(* CODESYS project Beer_machine.project

Project tree, tasks and I/O mapping:
  Device : CODESYS Control Win V3 x64, 3S - Smart Software Solutions GmbH, version 3.5.11.0
    application Application
      libraries: Standard, * (System); VisuDialogs, * (System); Util, * (System)
      task MainTask (cyclic, interval t#10ms, priority 1) calls Plant, Controller
      program Plant [ST]
      global variables GVL
      program Controller [ST]
      visualisation Visualization
      image pool ImagePool
  text list GlobalTextList
  5ce3da45-db07-42e7-a21c-a00fff4ed8f6|C:\Users\mihas\Documents\NSU2026\AM\images\input\MAX.png
  5ce3da45-db07-42e7-a21c-a00fff4ed8f6|C:\Users\mihas\Documents\NSU2026\AM\images\input\beer.png
  5ce3da45-db07-42e7-a21c-a00fff4ed8f6|C:\Users\mihas\Documents\NSU2026\AM\images\input\cigaretes after vki .png
  5ce3da45-db07-42e7-a21c-a00fff4ed8f6|C:\Users\mihas\Documents\NSU2026\AM\images\input\greencard.png
  5ce3da45-db07-42e7-a21c-a00fff4ed8f6|C:\Users\mihas\Documents\NSU2026\AM\images\input\jaguar.png
  5ce3da45-db07-42e7-a21c-a00fff4ed8f6|C:\Users\mihas\Documents\NSU2026\AM\images\input\monster.png
  5ce3da45-db07-42e7-a21c-a00fff4ed8f6|C:\Users\mihas\Documents\NSU2026\AM\images\input\pistol.png
  5ce3da45-db07-42e7-a21c-a00fff4ed8f6|C:\Users\mihas\Documents\NSU2026\AM\images\input\voenbilet.png
  5ce3da45-db07-42e7-a21c-a00fff4ed8f6|C:\Users\fish\AC_Beer_machine\img\input\blue monster.png
  5ce3da45-db07-42e7-a21c-a00fff4ed8f6|C:\Users\fish\AC_Beer_machine\img\input\monster.png
  5ce3da45-db07-42e7-a21c-a00fff4ed8f6|C:\Users\fish\AC_Beer_machine\img\input\red monster.jpg
  5ce3da45-db07-42e7-a21c-a00fff4ed8f6|C:\Users\fish\AC_Beer_machine\img\input\white monster.png
  5ce3da45-db07-42e7-a21c-a00fff4ed8f6|C:\Users\fish\AC_Beer_machine\img\input\yellow monster.png
*)

// Device/Application/GVL
VAR_GLOBAL
END_VAR

// Device/Application/Plant
PROGRAM Plant

VAR CONSTANT
	text_welcome_message : WSTRING(250) := "Здравстсвуйте!!!$nВыберите товар.";
	text_out_of_stock : WSTRING(250) := "Выбранного товара нет в наличии.$nПозвоните в поддержку, чтобы восполнить товар.";
	text_in_stock : WSTRING(250) := "Выбранный товар есть в наличии.$nПодготовка к оплате.";
	text_insert_payment : WSTRING(250) := "Оплатите товар.";
	text_not_enough_money : WSTRING(250) := "Внесите ещё.$nСредств недостаточно.";
	text_stuff_not_dropped : WSTRING(250) := "Товар не сбросился.$n Позвоните в поддержку, чтобы вернули деньги";
	text_mission_completed : WSTRING(250) := "Спасибо за покупку.$nНаслаждайтесь нашей продукцией!";
	
	text_arr : ARRAY[0..6] OF WSTRING(250) := [text_welcome_message, text_out_of_stock, text_in_stock, text_insert_payment, text_not_enough_money, text_stuff_not_dropped, text_mission_completed];
END_VAR

VAR
	cur : BOOL;
	dx : DINT;
	start_time_ms : DINT := TIME_TO_DINT(TIME());
	start_time_text : DINT := TIME_TO_DINT(TIME());
	start_time_angle : DINT := TIME_TO_DINT(TIME());
	angle : DINT := 0;
	j : DINT := 0;
	text_display : WSTRING(250);
	
	
	Drop_control : BOOL := 0;
	
	Drop_control1 : BOOL := 0;
	Drop_control2 : BOOL := 0;
	Drop_control3 : BOOL := 0;
	Drop_control4 : BOOL := 0;
	Drop_control5 : BOOL := 0;

	
	Spring1_prev : BOOL := 0;
	Spring2_prev : BOOL := 0;
	Spring3_prev : BOOL := 0;
	Spring4_prev : BOOL := 0;
	Spring5_prev : BOOL := 0;


	
	

END_VAR

VAR
	
	user: INT;
END_VAR

VAR
	MAX_call : BOOL;
	i : INT;
	
	tratit_bank : BOOL := FALSE;
	kopit_bank : BOOL := FALSE;
	user_bank : UDINT := 0;
	tovar : ARRAY[1..5] OF INT := [3, 3, 3, 3, 3];
END_VAR

// Поворот пружины
IF ((TIME_TO_DINT(TIME())) - start_time_angle) MOD 2000 > (1000 / 25) THEN 
	start_time_angle := TIME_TO_DINT(TIME());
	angle := (angle + 360 / 25) MOD 360;
END_IF

//взаимодействие с банком 
IF kopit_bank THEN
	user_bank := user_bank + 1;
	kopit_bank := FALSE;
END_IF
IF tratit_bank THEN
	IF user_bank > 0 THEN 
		user_bank := user_bank - 1;
	END_IF
	tratit_bank := FALSE;
END_IF

//датчики наличия товара

Controller.Obj1 := tovar[1] > 0;
Controller.Obj2 := tovar[2] > 0;
Controller.Obj3 := tovar[3] > 0;
Controller.Obj4 := tovar[4] > 0;
Controller.Obj5 := tovar[5] > 0;


//сброс товара

Drop_control1 := Controller.Spring1 AND NOT Spring1_prev;
Spring1_prev := Controller.Spring1;

Drop_control2 := Controller.Spring2 AND NOT Spring2_prev;
Spring2_prev := Controller.Spring2;

Drop_control3 := Controller.Spring3 AND NOT Spring3_prev;
Spring3_prev := Controller.Spring3;

Drop_control4 := Controller.Spring4 AND NOT Spring4_prev;
Spring4_prev := Controller.Spring4;

Drop_control5 := Controller.Spring5 AND NOT Spring5_prev;
Spring5_prev := Controller.Spring5;

Drop_control := Drop_control1 OR Drop_control2 OR Drop_control3 OR Drop_control4 OR Drop_control5;
Controller.Drop_control := Drop_control;

IF Drop_control1 THEN
	tovar[1] := MAX(tovar[1] - 1, 0);
END_IF
IF Drop_control2 THEN
		tovar[2] := MAX(tovar[2] - 1, 0);
END_IF
IF Drop_control3 THEN
		tovar[3] := MAX(tovar[3] - 1, 0);
END_IF
IF Drop_control4 THEN
		tovar[4] := MAX(tovar[4] - 1, 0);
END_IF
IF Drop_control5 THEN
		tovar[5] := MAX(tovar[5] - 1, 0);
END_IF


//пополнение товара
IF MAX_call THEN
	FOR i := 1 TO 5 DO
		tovar[i] := 3;
	END_FOR;
END_IF


//отображение текста по управляющему сигналу контроллера
text_display := text_arr[Controller.text_display_idx];

END_PROGRAM

// Device/Application/Controller
PROGRAM Controller

VAR_INPUT
	Obj1 : BOOL;
	Obj2 : BOOL;
	Obj3 : BOOL;
	Obj4 : BOOL;
	Obj5 : BOOL;
	Drop_control : BOOL;
	Button1 : BOOL;
	Button2 : BOOL;
	Button3 : BOOL;
	Button4 : BOOL;
	Button5 : BOOL;
	Cancellation : BOOL;
	bank_terminal : UDINT;
	cash_terminal : UDINT;
END_VAR

VAR_OUTPUT
	Spring1 : BOOL;
	Spring2 : BOOL;
	Spring3 : BOOL;
	Spring4 : BOOL;
	Spring5 : BOOL;
	text_display_idx : UDINT;
	credit : UDINT;
END_VAR

VAR CONSTANT
	price1 : UDINT := 15;
	price2 : UDINT := 10;
	price3 : UDINT := 5;
	price4 : UDINT := 7;
	price5 : UDINT := 20;
	_P_MAIN_LOOP_S_PRODUCT_CHOSING : INT := 0;
	_P_MAIN_LOOP_S_PAYMENT_WAIT : INT := 1;
	_P_MAIN_LOOP_S_INSERT_PAYMENT : INT := 2;
	_P_MAIN_LOOP_S_NOT_ENOUGH_MONEY : INT := 3;
	_P_MAIN_LOOP_S_GIVE_CHANGE : INT := 4;
	_P_MAIN_LOOP_S_NO_WAIT_CHANGE : INT := 5;
	_P_MAIN_LOOP_S_GIVE_PRODUCT : INT := 6;
	_P_MAIN_LOOP_S_GIVE_PRODUCT_TIMEOUT : INT := 7;
	_STOP : INT := 254;
	_ERROR : INT := 255;
END_VAR

VAR
	active_button : UDINT;
	cash_prev : UDINT;
	user_change : UDINT;
	_global_time : TIME;
	_g_p_Main_Loop_time : TIME;
	_g_p_Main_Loop_state : INT := _P_MAIN_LOOP_S_PRODUCT_CHOSING;
END_VAR

_global_time := TIME();

CASE _g_p_Main_Loop_state OF
	_P_MAIN_LOOP_S_PRODUCT_CHOSING:
		active_button := 0;
		cash_prev := 0;
		IF Cancellation THEN
			_g_p_Main_Loop_state := _P_MAIN_LOOP_S_NO_WAIT_CHANGE;
		END_IF
		IF Button1 THEN
			active_button := 1;
			IF NOT Obj1 THEN
				text_display_idx := 1;
			END_IF
			IF Obj1 THEN
				_g_p_Main_Loop_time := _global_time;
				_g_p_Main_Loop_state := _P_MAIN_LOOP_S_PAYMENT_WAIT;
			END_IF
		END_IF
		IF Button2 THEN
			active_button := 2;
			IF NOT Obj2 THEN
				text_display_idx := 1;
			END_IF
			IF Obj2 THEN
				_g_p_Main_Loop_time := _global_time;
				_g_p_Main_Loop_state := _P_MAIN_LOOP_S_PAYMENT_WAIT;
			END_IF
		END_IF
		IF Button3 THEN
			active_button := 3;
			IF NOT Obj3 THEN
				text_display_idx := 1;
			END_IF
			IF Obj3 THEN
				_g_p_Main_Loop_time := _global_time;
				_g_p_Main_Loop_state := _P_MAIN_LOOP_S_PAYMENT_WAIT;
			END_IF
		END_IF
		IF Button4 THEN
			active_button := 4;
			IF NOT Obj4 THEN
				text_display_idx := 1;
			END_IF
			IF Obj4 THEN
				_g_p_Main_Loop_time := _global_time;
				_g_p_Main_Loop_state := _P_MAIN_LOOP_S_PAYMENT_WAIT;
			END_IF
		END_IF
		IF Button5 THEN
			active_button := 5;
			IF NOT Obj5 THEN
				text_display_idx := 1;
			END_IF
			IF Obj5 THEN
				_g_p_Main_Loop_time := _global_time;
				_g_p_Main_Loop_state := _P_MAIN_LOOP_S_PAYMENT_WAIT;
			END_IF
		END_IF
		IF active_button <> 0 THEN
			_g_p_Main_Loop_time := _global_time;
		END_IF
		IF (_global_time - _g_p_Main_Loop_time) >= T#3s THEN
			text_display_idx := 0;
			_g_p_Main_Loop_time := _global_time;
		END_IF
	_P_MAIN_LOOP_S_PAYMENT_WAIT:
		text_display_idx := 2;
		IF (_global_time - _g_p_Main_Loop_time) >= T#3s THEN
			_g_p_Main_Loop_time := _global_time;
			_g_p_Main_Loop_state := _P_MAIN_LOOP_S_INSERT_PAYMENT;
		END_IF
	_P_MAIN_LOOP_S_INSERT_PAYMENT:
		text_display_idx := 3;
		IF Cancellation THEN
			_g_p_Main_Loop_state := _P_MAIN_LOOP_S_NO_WAIT_CHANGE;
		END_IF
		IF cash_terminal > 0 THEN
			IF cash_prev < cash_terminal THEN
				credit := credit + cash_terminal;
			END_IF
			IF active_button = 1 AND credit >= price1 THEN
				credit := credit - price1;
				_g_p_Main_Loop_time := _global_time;
				_g_p_Main_Loop_state := _P_MAIN_LOOP_S_GIVE_PRODUCT;
			END_IF
			IF active_button = 2 AND credit >= price2 THEN
				credit := credit - price2;
				_g_p_Main_Loop_time := _global_time;
				_g_p_Main_Loop_state := _P_MAIN_LOOP_S_GIVE_PRODUCT;
			END_IF
			IF active_button = 3 AND credit >= price3 THEN
				credit := credit - price3;
				_g_p_Main_Loop_time := _global_time;
				_g_p_Main_Loop_state := _P_MAIN_LOOP_S_GIVE_PRODUCT;
			END_IF
			IF active_button = 4 AND credit >= price4 THEN
				credit := credit - price4;
				_g_p_Main_Loop_time := _global_time;
				_g_p_Main_Loop_state := _P_MAIN_LOOP_S_GIVE_PRODUCT;
			END_IF
			IF active_button = 5 AND credit >= price5 THEN
				credit := credit - price5;
				_g_p_Main_Loop_time := _global_time;
				_g_p_Main_Loop_state := _P_MAIN_LOOP_S_GIVE_PRODUCT;
			END_IF
		ELSE
			IF active_button = 1 AND bank_terminal >= price1 THEN
				_g_p_Main_Loop_time := _global_time;
				_g_p_Main_Loop_state := _P_MAIN_LOOP_S_GIVE_PRODUCT;
			END_IF
			IF active_button = 2 AND bank_terminal >= price2 THEN
				_g_p_Main_Loop_time := _global_time;
				_g_p_Main_Loop_state := _P_MAIN_LOOP_S_GIVE_PRODUCT;
			END_IF
			IF active_button = 3 AND bank_terminal >= price3 THEN
				_g_p_Main_Loop_time := _global_time;
				_g_p_Main_Loop_state := _P_MAIN_LOOP_S_GIVE_PRODUCT;
			END_IF
			IF active_button = 4 AND bank_terminal >= price4 THEN
				_g_p_Main_Loop_time := _global_time;
				_g_p_Main_Loop_state := _P_MAIN_LOOP_S_GIVE_PRODUCT;
			END_IF
			IF active_button = 5 AND bank_terminal >= price5 THEN
				_g_p_Main_Loop_time := _global_time;
				_g_p_Main_Loop_state := _P_MAIN_LOOP_S_GIVE_PRODUCT;
			END_IF
		END_IF
		cash_prev := cash_terminal;
		IF (_global_time - _g_p_Main_Loop_time) >= T#5s THEN
			_g_p_Main_Loop_time := _global_time;
			_g_p_Main_Loop_state := _P_MAIN_LOOP_S_NOT_ENOUGH_MONEY;
		END_IF
	_P_MAIN_LOOP_S_NOT_ENOUGH_MONEY:
		text_display_idx := 4;
		IF (_global_time - _g_p_Main_Loop_time) >= T#1s THEN
			_g_p_Main_Loop_time := _global_time;
			_g_p_Main_Loop_state := _P_MAIN_LOOP_S_INSERT_PAYMENT;
		END_IF
	_P_MAIN_LOOP_S_GIVE_CHANGE:
		IF credit > 0 THEN
			user_change := user_change + credit;
		END_IF
		credit := 0;
		IF (_global_time - _g_p_Main_Loop_time) >= T#3s THEN
			_g_p_Main_Loop_time := _global_time;
			_g_p_Main_Loop_state := _P_MAIN_LOOP_S_PRODUCT_CHOSING;
		END_IF
	_P_MAIN_LOOP_S_NO_WAIT_CHANGE:
		IF credit > 0 THEN
			user_change := user_change + credit;
		END_IF
		credit := 0;
		_g_p_Main_Loop_time := _global_time;
		_g_p_Main_Loop_state := _P_MAIN_LOOP_S_PRODUCT_CHOSING;
	_P_MAIN_LOOP_S_GIVE_PRODUCT:
		text_display_idx := 6;
		IF active_button = 1 THEN
			Spring1 := 1;
		END_IF
		IF active_button = 2 THEN
			Spring2 := 1;
		END_IF
		IF active_button = 3 THEN
			Spring3 := 1;
		END_IF
		IF active_button = 4 THEN
			Spring4 := 1;
		END_IF
		IF active_button = 5 THEN
			Spring5 := 1;
		END_IF
		IF Drop_control THEN
			Spring1 := 0;
			Spring2 := 0;
			Spring3 := 0;
			Spring4 := 0;
			Spring5 := 0;
			_g_p_Main_Loop_time := _global_time;
			_g_p_Main_Loop_state := _P_MAIN_LOOP_S_GIVE_CHANGE;
		END_IF
		IF (_global_time - _g_p_Main_Loop_time) >= T#3s THEN
			Spring1 := 0;
			Spring2 := 0;
			Spring3 := 0;
			Spring4 := 0;
			Spring5 := 0;
			_g_p_Main_Loop_time := _global_time;
			_g_p_Main_Loop_state := _P_MAIN_LOOP_S_GIVE_PRODUCT_TIMEOUT;
		END_IF
	_P_MAIN_LOOP_S_GIVE_PRODUCT_TIMEOUT:
		IF (_global_time - _g_p_Main_Loop_time) >= T#10s THEN
			_g_p_Main_Loop_time := _global_time;
			_g_p_Main_Loop_state := _P_MAIN_LOOP_S_PRODUCT_CHOSING;
		END_IF
END_CASE

END_PROGRAM

// Device/Application/Visualization
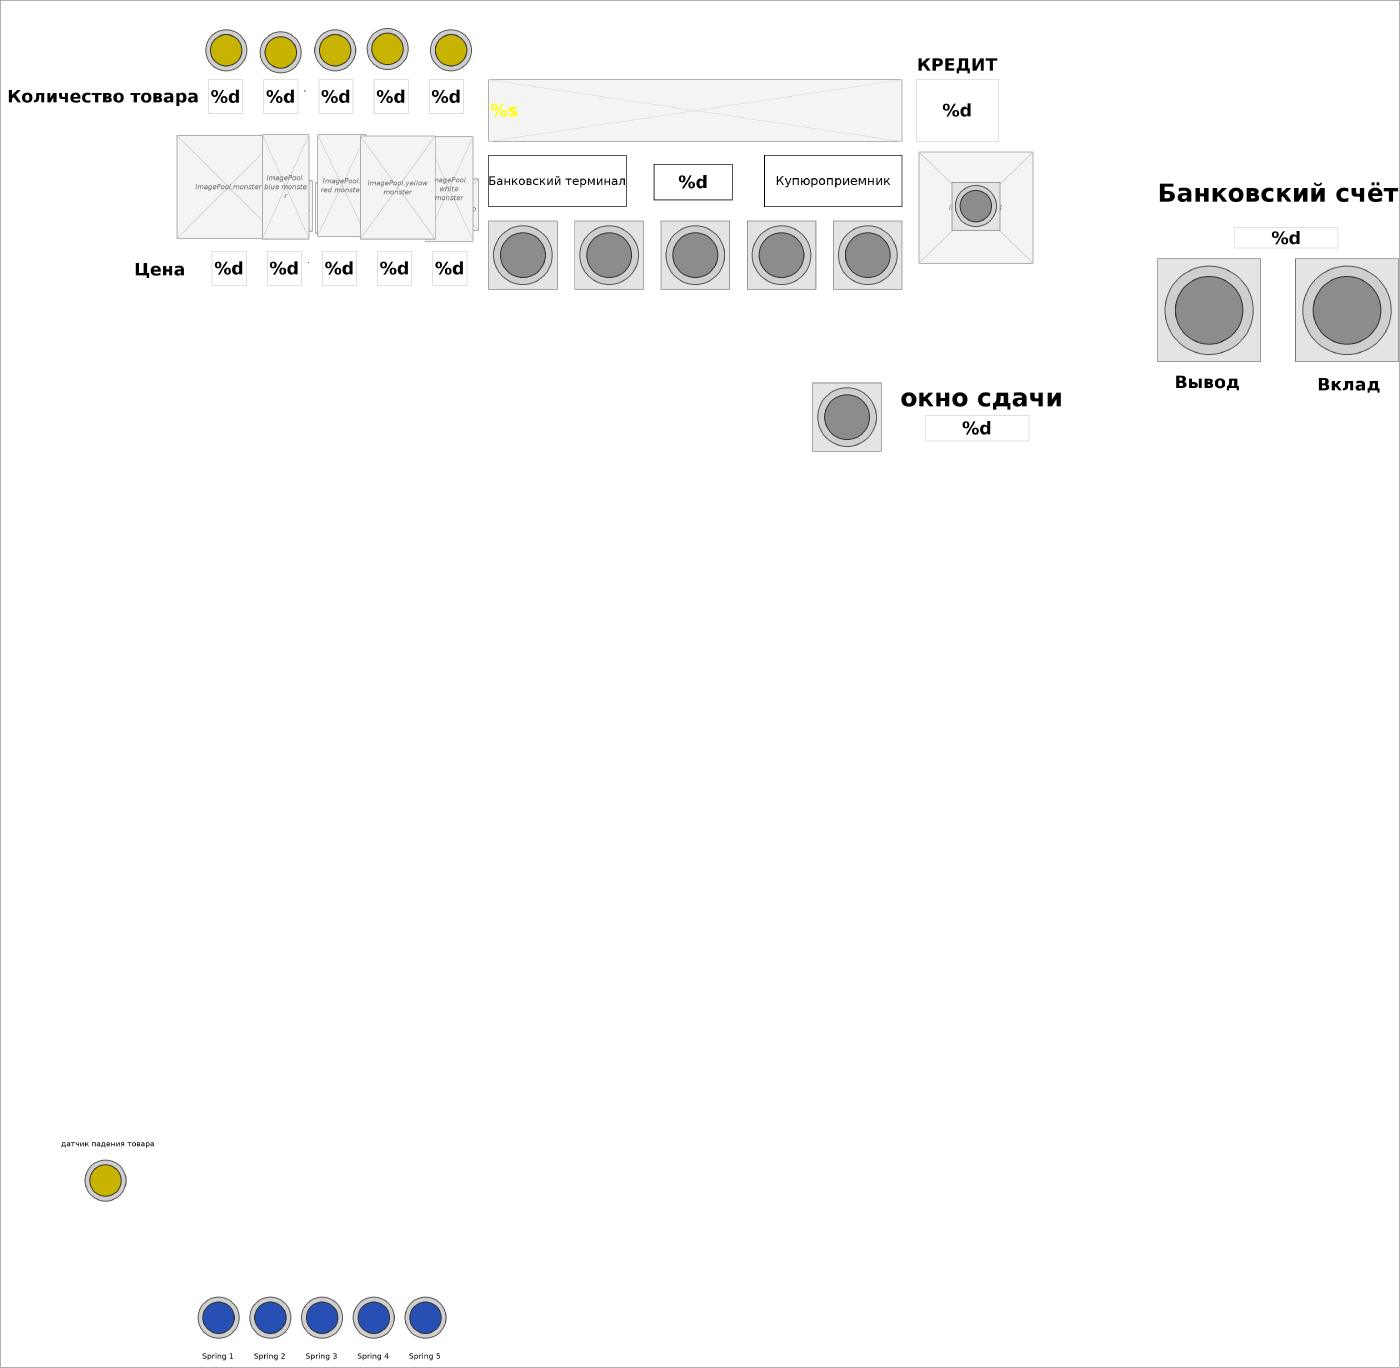
VISUALIZATION Visualization  // 2030x1985
    Polygon (441,131) (442,132)
    Lamp1 (282,1877 70x70), variable: Controller.Spring1, style: Lamp-Lamp1-Blue
    Lamp1 (357,1877 70x70), variable: Controller.Spring2, style: Lamp-Lamp1-Blue
    Lamp1 (432,1877 70x70), variable: Controller.Spring3, style: Lamp-Lamp1-Blue
    Lamp1 (507,1877 70x70), variable: Controller.Spring4, style: Lamp-Lamp1-Blue
    Lamp1 (582,1877 70x70), variable: Controller.Spring5, style: Lamp-Lamp1-Blue
    Image (708,115 600x90), "%s", tooltip "TIP TERMINAL", text variable: Plant.text_display, image: VisuDialogs.ImagePoolDialogs.Title
    Label (281,1953 70x30), "Spring 1"
    Label (581,1953 70x30), "Spring 5"
    Label (356,1953 70x30), "Spring 2"
    Label (431,1953 70x30), "Spring 3"
    Label (506,1953 70x30), "Spring 4"
    Image (295,262 75x75), image: ImagePool.spring_transp
    Image (619,259 75x75), image: ImagePool.spring_transp
    Image (378,261 75x75), image: ImagePool.spring_transp
    Image (457,264 75x75), image: ImagePool.spring_transp
    Image (541,259 75x75), image: ImagePool.spring_transp
    Lamp1 (118,1678 70x70), variable: Plant.Drop_control, style: Lamp-Lamp1-Yellow
    Label (85,1633 143x54), "датчик падения товара"
    Lamp1 (293,38 70x70), variable: Controller.Obj1, style: Lamp-Lamp1-Yellow
    Lamp1 (372,41 70x70), variable: Controller.Obj2, style: Lamp-Lamp1-Yellow
    Lamp1 (451,38 70x70), variable: Controller.Obj3, style: Lamp-Lamp1-Yellow
    Lamp1 (527,36 70x70), variable: Controller.Obj4, style: Lamp-Lamp1-Yellow
    Lamp1 (619,38 70x70), variable: Controller.Obj5, style: Lamp-Lamp1-Yellow
    Image (256,196 150x150), image: ImagePool.monster
    Textfield (302,115 50x50), "%d", text variable: Plant.tovar[1]
    Textfield (382,115 50x50), "%d", text variable: Plant.tovar[2]
    Textfield (462,115 50x50), "%d", text variable: Plant.tovar[3]
    Textfield (542,115 50x50), "%d", text variable: Plant.tovar[4]
    Textfield (622,115 50x50), "%d", text variable: Plant.tovar[5]
    PushSwitch (708,320 100x100), tooltip "1. платно?", variable: Controller.Button1, behaviour: TAP, style: Switch-PushSwitch-Gray
    PushSwitch (833,320 100x100), tooltip "2. платно?", variable: Controller.Button2, behaviour: TAP, style: Switch-PushSwitch-Gray
    PushSwitch (1208,320 100x100), tooltip "5. платно?", variable: Controller.Button5, behaviour: TAP, style: Switch-PushSwitch-Gray
    PushSwitch (1083,320 100x100), tooltip "4. платно?", variable: Controller.Button4, behaviour: TAP, style: Switch-PushSwitch-Gray
    PushSwitch (958,320 100x100), tooltip "3. платно?", variable: Controller.Button3, behaviour: TAP, style: Switch-PushSwitch-Gray
    PushSwitch (1178,555 100x100), tooltip "Отмена/Сдача", variable: Controller.Cancellation, behaviour: TAP, style: Switch-PushSwitch-Gray
    Label (1678,255 350x50), "Банковский счёт"
    Textfield (1790,330 150x30), "%d", text variable: Plant.user_bank
    PushSwitch (1878,375 150x150), tooltip "Вложить 1", variable: Plant.kopit_bank, behaviour: TOGGLE, style: Switch-PushSwitch-Gray
    Label (1909,535 94x45), "Вклад"
    PushSwitch (1678,375 150x150), tooltip "Снять 1", variable: Plant.tratit_bank, behaviour: TOGGLE, style: Switch-PushSwitch-Gray
    Label (1679,535 143x38), "Вывод"
    Label (1328,75 120x37), "КРЕДИТ"
    Rectangle (708,225 200x75), "Банковский терминал", tooltip "Приложить болт"
        OnMouseLeave: execute { Controller.bank_terminal := 0; }
        OnMouseEnter: execute { Controller.bank_terminal := Plant.user_bank; }
    Rectangle (1108,225 200x75), "Купюроприемник", tooltip "Поставить 5"
        OnMouseDown: execute { Controller.cash_terminal := 5; }
        OnMouseUp: execute { Controller.cash_terminal := 0; }
    Textfield (1328,115 120x90), "%d", text variable: Controller.credit
    Textfield (1341,602 151x38), "%d", tooltip "забрать сдачу", text variable: Controller.user_change
        OnMouseClick: execute { Controller.user_change := 0; }
    Label (1293,541 261x72), "окно сдачи"
    Image (1332,220 166x162), tooltip "звонок в поддержку", image: ImagePool.MAX
    PushSwitch (1380,264 70x70), tooltip "*только в MAX", variable: Plant.MAX_call, behaviour: TAP, style: Switch-PushSwitch-Gray
    Label (1331,322 166x54)
    Label (11,119 277x41), "Количество товара"
    Rectangle (948,238 114x52), "%d", tooltip "Выбранный товар", text variable: Controller.active_button
    Polygon (446,380) (447,381)
    Textfield (307,364 50x50), "%d", text variable: Controller.price1
    Textfield (387,364 50x50), "%d", text variable: Controller.price2
    Textfield (467,364 50x50), "%d", text variable: Controller.price3
    Textfield (547,364 50x50), "%d", text variable: Controller.price4
    Textfield (627,364 50x50), "%d", text variable: Controller.price5
    Label (170,370 124x41), "Цена"
    Image (380,195 68x152), image: ImagePool.blue monster
    Image (460,195 71x148), image: ImagePool.red monster
    Image (616,198 70x152), image: ImagePool.white monster
    Image (522,197 109x150), image: ImagePool.yellow monster
END_VISUALIZATION
